TYPE ST_AlarmenDepalletizer :
STRUCT
	Source : STRING(30);
	Timestamp : TIMESTRUCT;
	Text : STRING(80);
	Active : BOOL;
END_STRUCT
END_TYPE

(* stored: Version 1.1.0.1
   DUT ST_AlarmenDepalletizer: Id {98146235-5f66-4aa4-851b-b95e9e119467} *)
